FUNCTION_BLOCK LIFTER_XFER (* Lifter Pallet Transfer and Fault Simulation Logic *)
  (* Standard: 61499-2 *)
  (* Version 0.3, 2005-06-01, JHC, Holobloc Inc, Made REQ=>START mutually exclusive with others. *)
  (* Version 0.2, 2005-06-01, JHC, Holobloc Inc, Re-compiled with new emitter. *)
  (* Version 0.1, 2004-11-12, JHC, Rockwell Automation, Added FFLT, LFLT, TFLT and associated logic. *)
  (* Version 0.0, 2004-11-11, JHC, Rockwell Automation, Combined LIFTER_LDU and LIFTER_FAULT. *)
  (* Compiler header: package fb.rt.mach; *)
  (* Compiler Java Sun JDK 1.4.2 *)
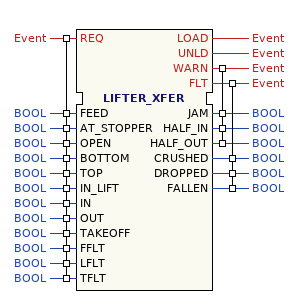
  EVENT_INPUT
    REQ WITH FEED, OPEN, BOTTOM, IN, OUT, AT_STOPPER, IN_LIFT, TOP, TAKEOFF, LFLT, FFLT, TFLT; (* Input Change Notification *)
  END_EVENT
  EVENT_OUTPUT
    LOAD; (* Load Lifter *)
    UNLD; (* Unload Lifter *)
    WARN WITH HALF_IN, JAM, HALF_OUT; (* Non-Fatal Fault Warning *)
    FLT WITH CRUSHED, FALLEN, DROPPED; (* Fatal Fault Notification *)
  END_EVENT
  VAR_INPUT
    FEED : BOOL; (* Feed Conveyor Motor ON *)
    AT_STOPPER : BOOL; (* Pallet at Stopper Position *)
    OPEN : BOOL; (* Stopper/Gate Open *)
    BOTTOM : BOOL; (* Lift at Bottom Position *)
    TOP : BOOL; (* Lift at Top Position *)
    IN_LIFT : BOOL; (* Pallet in Lift *)
    IN : BOOL; (* Lift Conveyor IN motor ON *)
    OUT : BOOL; (* Lift Conveyor OUT motor ON *)
    TAKEOFF : BOOL; (* Takeoff Conveyor Motor ON *)
    FFLT : BOOL; (* Feed Conveyor Fault *)
    LFLT : BOOL; (* Simulated Lifter Fault injected from UI *)
    TFLT : BOOL; (* Takeoff Conveyor Fault *)
  END_VAR
  VAR_OUTPUT
    JAM : BOOL; (* Jam at Lifter Entrance *)
    HALF_IN : BOOL; (* Bottom Pallet Half In Lifter *)
    HALF_OUT : BOOL;
    CRUSHED : BOOL; (* Crushed or Dropped *)
    DROPPED : BOOL;
    FALLEN : BOOL;
  END_VAR
  VAR
    FCOND : BOOL; (* Fault Condition *)
    WCOND : BOOL; (* Warning Condition *)
    LCOND : BOOL; (* LOAD condition *)
    UCOND : BOOL; (* UNLD condition *)
  END_VAR
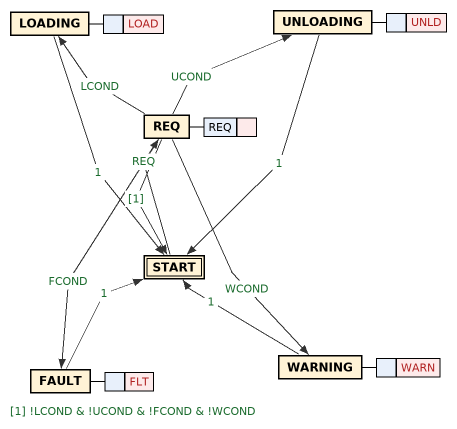
  EC_STATES
    START; (* Initial State *)
    REQ : REQ; (* Normal execution *)
    FAULT : -> FLT;
    WARNING : -> WARN;
    LOADING : -> LOAD;
    UNLOADING : -> UNLD;
  END_STATES
  EC_TRANSITIONS
    START TO REQ := REQ;
    REQ TO FAULT := FCOND;
    REQ TO WARNING := WCOND;
    REQ TO LOADING := LCOND;
    REQ TO UNLOADING := UCOND;
    REQ TO START := !LCOND & !UCOND & !FCOND & !WCOND;
    FAULT TO START := 1;
    WARNING TO START := 1;
    LOADING TO START := 1;
    UNLOADING TO START := 1;
  END_TRANSITIONS
  ALGORITHM REQ IN LD: (* Lifter Loading Physical Logic *)
    LCOND := FEED FFLT ! & AT_STOPPER & OPEN & BOTTOM & IN_LIFT ! & IN & OUT ! & LFLT ! &;
    UCOND := TOP IN_LIFT & OUT & IN ! & LFLT ! & TAKEOFF & TFLT ! &;
    JAM := FFLT ! FEED & AT_STOPPER & OPEN & BOTTOM & IN_LIFT &;
    CRUSHED := HALF_IN BOTTOM ! &;
    HALF_IN := FEED FFLT ! & AT_STOPPER & OPEN & BOTTOM & IN_LIFT ! & IN ! LFLT | &;
    DROPPED := FEED FFLT ! & AT_STOPPER & OPEN & BOTTOM ! & CRUSHED ! &;
    FALLEN := HALF_OUT TOP ! &;
    HALF_OUT := TOP IN_LIFT & OUT & IN ! & LFLT ! & TAKEOFF !  TFLT | &;
    FCOND := CRUSHED DROPPED | FALLEN |;
    WCOND := JAM HALF_IN | HALF_OUT |;
  END_ALGORITHM
END_FUNCTION_BLOCK
